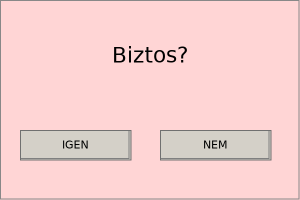
VISUALIZATION Biztos  // 300x200
    Label (10,40 281x30), "Biztos?"
    Button (20,130 111x30), "IGEN"
        toggle GVL.Biztos
        OnMouseClick: CloseDialog Dialog=Biztos, Result=OK, NumpadKeypadSet=True
    Button (160,130 111x30), "NEM"
        OnMouseClick: CloseDialog Dialog=Biztos, Result=OK, NumpadKeypadSet=True
END_VISUALIZATION

(* stored: Version 1.1.0.1, ProductVersion 3.1.4024.11
   Visu Biztos: Id {319bf461-45ce-4e2e-9e4a-6def5ad6c50f} *)
